# EPICS substitutions: utcaApp/Db/fmc_active_clk.substitutions
file db/scan_task.template {
    {}
}

file db/fmc_active_clk.template {
    {}
}
